FUNCTION_BLOCK aiIntToVtqReal (* Converte valor bruto INT (remota) em VTQREAL para a entrada externa do aiSignalDecode *)
  (* Standard: 61499-2 *)
  (* Version 1.0, 10/5/2026, Hidryco, Hidryco, Entrada INT para AnalogInput (4-20 mA via TM3BCEIP) *)
  PACKAGE SE.Nereda;
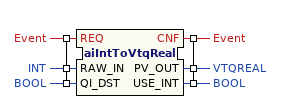
  EVENT_INPUT
    REQ WITH RAW_IN, QI_DST; (* Novo valor bruto *)
  END_EVENT
  EVENT_OUTPUT
    CNF WITH PV_OUT, USE_INT; (* Valor convertido *)
  END_EVENT
  VAR_INPUT
    RAW_IN : INT; (* Valor bruto do canal (symlink AInInt) *)
    QI_DST : BOOL; (* QO do SYMLINKMULTIVARDST (TRUE = symlink conectado) *)
  END_VAR
  VAR_OUTPUT
    PV_OUT : VTQREAL; (* Valor bruto em VTQREAL *)
    USE_INT : BOOL; (* TRUE = usar a entrada INT no lugar do rawPv *)
  END_VAR
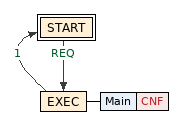
  EC_STATES
    START; (* Initial State *)
    EXEC : Main -> CNF;
  END_STATES
  EC_TRANSITIONS
    START TO EXEC := REQ;
    EXEC TO START := 1;
  END_TRANSITIONS
  ALGORITHM Main IN ST: (* Conversao INT para VTQREAL *)
(* Converte o valor bruto INT de um canal analogico de remota (TM3AI8 via Modbus)
   em VTQREAL para a entrada externa do aiSignalDecode. USE_INT so vai para TRUE quando o
   symlink AInInt esta efetivamente conectado (QO do SYMLINKMULTIVARDST). *)
IF QI_DST THEN
    PV_OUT.value := INT_TO_REAL(RAW_IN);
    PV_OUT.quality := 16#00000000;
    USE_INT := TRUE;
END_IF;
  END_ALGORITHM
END_FUNCTION_BLOCK
